TYPE (* Human readable text with an optional locale identifier *)
  (* Standard: 61499-2 *)
  (* Version 1.0, 2019-07-08, Jose Cabral, fortiss GmbH *)
  (* ASN.1 tag APPLICATION 1 *)
  LocalizedText : STRUCT
    text : STRING; (* The localized text *)
    locale : STRING; (* The identifier for the locale (e.g. "en-US"). *)
  END_STRUCT;
END_TYPE
